// TIA Portal V18 export
TYPE "MEStoPLC_MainCheckOut"
// stored: IsFailsafeCompliant false
   STRUCT
      "M-DataSaveDone" : Bool;   // 过程数据采集完成标志位，此信号串入放行逻辑，MES置位后PLC立即复位请求数据采集信号P-DataReady，P-DataReady下降沿由MES复位此信号
      "M-DataSaveOK" : Bool;   // 工件可加工标志位，PLC收到M-ReqMesDone+此信号后可开始加工
      "M-DataSaveNG" : Bool;   // 工件可不加工标志位，PLC收到M-ReqMesDone+此信号后可放行
      "M-DataSaveErrCode" : Int;   // 【预留】“M-ErrorMsg”失效的时候启用
      "M-DataSaveErrMsg" : String[98];   // P-ReqMes请求Mes标志位收到后，如果Mes对请求的数据校验有异常，写入相应中文字符串，M-ReqMesDone信号超时后将中文字符串显示到HMI
      Reserve : Array[1..2096] of Byte;   // CheckOut预留
   END_STRUCT;
END_TYPE
